// Mitsubishi GX Works2 project: 水塔水位模拟控制   PLC: FX1S

PROGRAM MAIN
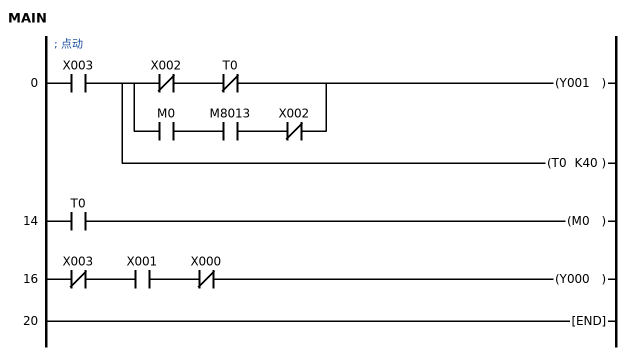
; 点动
0     LD      X003
      MPS
      LDI     X002
      ANI     T0
      LD      M0
      AND     M8013
      ANI     X002
      ORB
      ANB
      OUT     Y001
      MPP
      OUT     T0 K40
14    LD      T0
      OUT     M0
16    LDI     X003
      AND     X001
      ANI     X000
      OUT     Y000
20    END
END_PROGRAM
